(* IEC 61131-3 sources: brdkVision/export/brdkViBase/V1.00.3, 2 files *)

(* ---- Types.typ ---- *)
TYPE
	brdkViBase_hw_in_common_typ : 	STRUCT  (*B&R common hardware input structure from device*)
		hardwareVariant : UDINT; (*The hardware variant of the module can be read from this data point.*)
		moduleId : UDINT; (*The module hardware ID used to determine the type of device that can be read from this register. This is also listed in the respective technical data as the "B&R ID code". In addition, a serial number is printed on each module; the module hardware ID corresponds to the first four positions of this serial number.*)
		firmwareVersion : UDINT; (*The firmware version of the module can be read from this data point.
The last two positions correspond to the number after the decimal point.
Example: 345 corresponds to version 3.45.*)
		serialNumber : UDINT; (*The module's unique serial number can be read from this register. This 7-digit serial number is printed in decimal form on the module's housing*)
		moduleOk : BOOL; (*Status bit that indicates whether the module is physically present and configured. Detection takes place via the Fieldbus connection.*)
	END_STRUCT;
	brdkViBase_2d_typ : 	STRUCT  (*2D vector information.*)
		y : LREAL; (*Y-coordinate.*)
		x : LREAL; (*X-coordinate.*)
	END_STRUCT;
	brdkViBase_3d_typ : 	STRUCT  (*3D vector information.*)
		y : LREAL; (*Y-coordinate.*)
		z : LREAL; (*Z-coordinate.*)
		x : LREAL; (*X-coordinate.*)
	END_STRUCT;
	brdkViBase_angle_enum :
		( (*Angle enumeration type.*)
		BRDKVIBASE_ANGLE_X, (*X-angle*)
		BRDKVIBASE_ANGLE_Y, (*Y-angle*)
		BRDKVIBASE_ANGLE_Z (*Z-angle*)
		);
END_TYPE

(*Hw for camera *)

TYPE
	brdkViBase_cam_hw_out_typ : 	STRUCT  (*Camera hardware output structure to device*)
		par : brdkViBase_cam_hw_out_par_typ; (*Hardware output parameters to the device*)
		cmd : brdkViBase_cam_hw_out_cmd_typ; (*Hardware out commands to the device*)
	END_STRUCT;
	brdkViBase_cam_hw_out_cmd_typ : 	STRUCT  (*Camera hardware command structure to device*)
		imageAcquisition : BOOL; (*Enables/Disables the trigger for the image acquisition*)
		resetAcquisiton : BOOL; (*Cancels an image acquisition triggered by NetTime*)
		searchAcquisitonSettings : BOOL; (*Enables/Disables search for focus and integration time of the sensor*)
		digitalOutput : BOOL; (*Selects the mode of operation of the digital output*)
	END_STRUCT;
	brdkViBase_cam_hw_out_par_typ : 	STRUCT  (*Camera hardware parameter structure to device*)
		statusLED : USINT; (*Selects the mode and color of the LED status indicator bars. Constants BRDKVIBASE_STATUS_xxx can be used to set the color*)
		gainLevel : USINT; (*Sets a gain factor*)
		focus : UINT; (*Sets the focus from "MOD" to "Infinity", Unit depends on the selected one in the vision application file (um, mm, raw)*)
		exposureTime : UDINT; (*Sets the integration time of the sensor in microseconds*)
		flashColor : USINT; (*Selects LED colors of the onboard LED lighting. The constants BRDKVIBASE_LED_xxx can be used to set the color*)
		flashSegment : USINT; (*Enables/Disables LED segments. Binary patter for enable each of the four segments 0000 = all off, 1111 = all on*)
		chromaticLock : BOOL; (*Enables/Disables ChromaticLock*)
		IRFilter : BOOL; (*Enables/Disables the infrared filter*)
		delayNetTime : DINT; (*Sets Delay or NetTime for the trigger in microseconds*)
		cyclicLineScanPeriod : DINT; (*Time between 2 image acquisitions in dynamic line sensor operation.*)
		cyclicLineScanNettime : DINT; (*Specifies the NetTime for dynamic line sensor mode.*)
	END_STRUCT;
	brdkViBase_cam_hw_in_status_typ : 	STRUCT  (*Camera hardware status input structure from device*)
		sensorTemperature : SINT; (*Current camera temperature in °C*)
		lightWarningCnt : USINT; (*Counter for errors or warnings that have occurred related to lighting.*)
		cameraStatus : UDINT; (*This parameter specifies the status of the camera.*)
		acceptedAcquisitionCnt : USINT; (*Counter for accepted image acquisitions*)
		completedAcquisitionCnt : USINT; (*Counter for performed image acquisitions*)
		failedAcquisitionCnt : USINT; (*Counter for failed image acquisitions*)
		undervoltageError : BOOL; (*Power supply alarm*)
		imageAcquisitionReady : BOOL; (*Camera availability status*)
		imageProcessingActive : BOOL; (*Status of image processing execution *)
		digitalOutputStatus : BOOL; (*Status of digital output 01*)
		cameraProcessingTime : UINT; (*Processing time in milliseconds*)
		imageProcessingError : UINT; (*Bit pattern for displaying errors and warnings that occurred during image processing.*)
		imageNettime : DINT; (*NetTime of the image in microseconds*)
		digitalInput : BOOL; (*Status digital input (trigger input)*)
		gainLevel : USINT; (*Current GainLevel*)
		focus : UINT; (*Current focus setting from "MOD" to "Infinity", Unit depends on the selected one in the vision application file (um, mm, raw)*)
		exposureTime : UDINT; (*Current integration time of the sensor in microseconds *)
	END_STRUCT;
	brdkViBase_cam_hw_in_typ : 	STRUCT  (*Camera hardware input structure from device*)
		common : brdkViBase_hw_in_common_typ; (*B&R Hardware common inputs from device*)
		status : brdkViBase_cam_hw_in_status_typ; (*Camera hardware status inputs from device*)
	END_STRUCT;
	brdkViBase_cam_hw_typ : 	STRUCT  (*Camera hardware structure*)
		in : brdkViBase_cam_hw_in_typ; (*Camera hardware inputs from device*)
		out : brdkViBase_cam_hw_out_typ; (*Camera hardware outputs to device*)
	END_STRUCT;
END_TYPE

(*hw for light*)

TYPE
	brdkViBase_light_hw_out_typ : 	STRUCT  (*Light hardware output structure to device*)
		cmd : brdkViBase_light_hw_out_cmd_typ; (*Light hardware output commands to device*)
		par : brdkViBase_light_hw_out_par_typ; (*Light hardware output parameters to device*)
	END_STRUCT;
	brdkViBase_light_hw_status_typ : 	STRUCT  (*Light hardware status structure from device*)
		ready : BOOL; (*Lighting unit availability status*)
		status : UDINT; (*This parameter specifies the status of the lighting unit.*)
		acceptedFlashCnt : USINT; (*Counter for accepted lighting jobs*)
		completedFlashCnt : USINT; (*Counter for executed lighting jobs*)
		failedFlashCnt : USINT; (*Counter for failed lighting jobs*)
		LightWarningCnt : USINT; (*Counter for errors or warnings that have occurred related to lighting.*)
		sensorTemperature : SINT; (*Current lighting unit temperature in °C*)
	END_STRUCT;
	brdkViBase_light_hw_in_typ : 	STRUCT  (*Light hardware input structure from device*)
		common : brdkViBase_hw_in_common_typ; (*B&R hardware common inputs from device*)
		status : brdkViBase_light_hw_status_typ; (*Light hardware status inputs from device*)
	END_STRUCT;
	brdkViBase_light_hw_typ : 	STRUCT  (*Light hardware structure*)
		in : brdkViBase_light_hw_in_typ; (*Light hardware inputs from device*)
		out : brdkViBase_light_hw_out_typ; (*Light hardware outputs to device*)
	END_STRUCT;
	brdkViBase_light_hw_out_cmd_typ : 	STRUCT  (*Light hardware output commands to device*)
		flashTrigger : BOOL; (*Enables/Disables the trigger for the lighting job*)
		resetFlashTrigger : BOOL; (*Canceling a lighting job triggered by NetTime*)
	END_STRUCT;
	brdkViBase_light_hw_out_par_typ : 	STRUCT  (*Light hardware parameter output structure to device*)
		flashColor : USINT; (*Select LED colors of the LED lighting
 Constant BRDKVIBASE_LED_xxx can be used to set the color*)
		exposureTime : UDINT; (*Sets the exposure time in µs*)
		flashAngle : USINT; (*Only for Lightbar. Position of the stepper motor in degree 0 to 135*)
		flashSegments : USINT; (*Only for Lightbar. Enables/Disables LED segments*)
		cyclicLineScanPeriod : DINT; (*Time between 2 flashes in dynamic line sensor operation.*)
		cyclicLineScanNettime : DINT; (*Specifies the NetTime for dynamic line sensor mode.*)
		nettime : DINT; (*Sets the NetTime for the trigger in µs*)
	END_STRUCT;
END_TYPE

(*hw for vision function*)

TYPE
	brdkviBase_hw_vf_out_offset_typ : 	STRUCT  (*Offset ROI outputs for vision functions*)
		x : DINT; (*Offset of the ROI in the x-direction in 1/100 pixel increments.*)
		y : DINT; (*Offset of the ROI in the y-direction in increments of 1/100 pixel.*)
		orientation : INT; (*Offset to orient the ROI from -179.99° to +180° in 1/100 degree steps*)
		rotCenterX : DINT; (*Offset to orient the ROI from -179.99° to +180° in 1/100 degree steps*)
		rotCenterY : DINT; (*Offset of the rotation center in the y-direction in increments of 1/100 pixel.*)
	END_STRUCT;
	brdkViBase_hw_vf_in_common_typ : 	STRUCT  (*Common vision function hardware input structure from device*)
		numResults : USINT; (*Number of results found*)
		functionProcessingTime : UINT; (*Processing time of the visual function in microseconds*)
	END_STRUCT;
	brdkViBase_hw_vf_out_common_typ : 	STRUCT  (*vision function hardware output structure to device*)
		enable : BOOL; (*Enables/Disables the function*)
		numSearchMax : USINT; (*Maximum number of codes to search*)
		alignment : USINT; (*0 = "None"
1 = "SetReference"
2 = "GenerateAlignmentData" *)
		offsetROI : brdkviBase_hw_vf_out_offset_typ; (*Offset ROI parameters*)
	END_STRUCT;
END_TYPE

(*VF BLOB*)

TYPE
	brdkViBase_hw_blob_out_typ : 	STRUCT  (*BLOB hardware output structure*)
		regionFeatures : BOOL; (*Enables the geometric exclusion procedure *)
		enhancedBlobInformation : BOOL; (*0 = Additional information is transferred (default).
1 = Additional information is not transferred.
Means an increase of FunctionProcessingTime *)
		common : brdkViBase_hw_vf_out_common_typ; (*Common vision function output*)
	END_STRUCT;
	brdkViBase_hw_blob_in_typ : 	STRUCT  (*BLOB hardware structure for a result*)
		modelNumber : USINT; (*ModelNumber of the found blob*)
		meanGreyValue : USINT; (*Arithmetic mean of grayscale values for the blob*)
		clipped : BOOL; (* Edge contact detection *)
		area : UDINT; (* Size (area) in pixels in increments of 1/100 pixel*)
		length : UDINT; (* Length of the found blob*)
		width : UDINT; (* Width of the found blob. Is always the longer of the two sides*)
		xMin : DINT; (* Extreme value in the column direction
Minimum column position of the BLOB area*)
		xMax : DINT; (*Extreme value in the column direction
Maximum column position of the BLOB area*)
		yMin : DINT; (*Extreme value in the line direction
Minimum line position of the BLOB area*)
		yMax : DINT; (*Extreme value in the line direction
Maximum line position of the BLOB area*)
		circularity : USINT; (*Circularity of the found blob in %*)
		rectangularity : USINT; (*Rectangularity of the found blob in %*)
		anisometry : UINT; (*Anisometry of the found blob*)
		innterCirclePositionX : DINT; (*Output of position X of the center point of the inner circle of the found blob determined by the algorithm in 1/100 pixels.*)
		innterCirclePositionY : DINT; (*Output of position Y of the center point of the inner circle of the found blob determined by the algorithm in 1/100 pixels.*)
		innterCircleRadius : UDINT; (*Output of the radius of the inner circle of the found blob determined by the algorithm in 1/100 pixels.*)
		positionX : DINT; (*X-position (of the found blob) in the image in increments of 1/100 pixel*)
		positionY : DINT; (*Y-position (of the found blob) in the image in increments of 1/100 pixel*)
		orientation : INT; (*-179.99° to +180° in increments of 1/100 degree*)
		rotCenterX : DINT; (*The value deviating from the specified taught-in Alignment model is output here. In 1/100 pixel steps*)
		rotCenterY : DINT; (*The value deviating from the specified taught-in Alignment model is output here. In 1/100 pixel steps*)
	END_STRUCT;
	brdkViBase_hw_blob_1_in_typ : 	STRUCT  (*BLOB hardware input structure for 1 BLOB result*)
		common : brdkViBase_hw_vf_in_common_typ;
		results : brdkViBase_hw_blob_in_typ;
	END_STRUCT;
	brdkViBase_hw_blob_1_typ : 	STRUCT  (*BLOB hardware structure for 1 BLOB result*)
		in : brdkViBase_hw_blob_1_in_typ;
		out : brdkViBase_hw_blob_out_typ;
	END_STRUCT;
	brdkViBase_hw_blob_10_in_typ : 	STRUCT  (*BLOB hardware input structure for 10 BLOB result*)
		common : brdkViBase_hw_vf_in_common_typ;
		results : ARRAY[0..9]OF brdkViBase_hw_blob_in_typ;
	END_STRUCT;
	brdkViBase_hw_blob_10_typ : 	STRUCT  (*BLOB hardware structure for 10 BLOB result*)
		in : brdkViBase_hw_blob_10_in_typ;
		out : brdkViBase_hw_blob_out_typ;
	END_STRUCT;
	brdkViBase_hw_blob_50_in_typ : 	STRUCT  (*BLOB hardware input structure for 50 BLOB result*)
		common : brdkViBase_hw_vf_in_common_typ;
		results : ARRAY[0..49]OF brdkViBase_hw_blob_in_typ;
	END_STRUCT;
	brdkViBase_hw_blob_50_typ : 	STRUCT  (*BLOB hardware structure for 50 BLOB result*)
		in : brdkViBase_hw_blob_10_in_typ;
		out : brdkViBase_hw_blob_out_typ;
	END_STRUCT;
	brdkViBase_hw_blob_100_in_typ : 	STRUCT  (*BLOB hardware input structure for 100 BLOB result*)
		common : brdkViBase_hw_vf_in_common_typ;
		results : ARRAY[0..99]OF brdkViBase_hw_blob_in_typ;
	END_STRUCT;
	brdkViBase_hw_blob_100_typ : 	STRUCT  (*BLOB hardware structure for 100 BLOB result*)
		in : brdkViBase_hw_blob_100_in_typ;
		out : brdkViBase_hw_blob_out_typ;
	END_STRUCT;
	brdkViBase_hw_blob_150_in_typ : 	STRUCT  (*BLOB hardware input structure for 150 BLOB result*)
		common : brdkViBase_hw_vf_in_common_typ;
		results : ARRAY[0..149]OF brdkViBase_hw_blob_in_typ;
	END_STRUCT;
	brdkViBase_hw_blob_150_typ : 	STRUCT  (*BLOB hardware structure for 150 BLOB result*)
		in : brdkViBase_hw_blob_150_in_typ;
		out : brdkViBase_hw_blob_out_typ;
	END_STRUCT;
	brdkViBase_hw_blob_200_in_typ : 	STRUCT  (*BLOB hardware input structure for 200 BLOB result*)
		common : brdkViBase_hw_vf_in_common_typ;
		results : ARRAY[0..199]OF brdkViBase_hw_blob_in_typ;
	END_STRUCT;
	brdkViBase_hw_blob_200_typ : 	STRUCT  (*BLOB hardware structure for 200 BLOB result*)
		in : brdkViBase_hw_blob_200_in_typ;
		out : brdkViBase_hw_blob_out_typ;
	END_STRUCT;
	brdkViBase_hw_blob_250_in_typ : 	STRUCT  (*BLOB hardware input structure for 250 BLOB result*)
		common : brdkViBase_hw_vf_in_common_typ;
		results : ARRAY[0..249]OF brdkViBase_hw_blob_in_typ;
	END_STRUCT;
	brdkViBase_hw_blob_250_typ : 	STRUCT  (*BLOB hardware structure for 250 BLOB result*)
		in : brdkViBase_hw_blob_250_in_typ;
		out : brdkViBase_hw_blob_out_typ;
	END_STRUCT;
END_TYPE

(*VF match*)

TYPE
	brdkViBase_hw_match_out_typ : 	STRUCT  (*Matching hardware output structure*)
		timeout : UINT; (*Time limit for the search time in increments of 1 ms. 0 = no timeout*)
		minScore : USINT; (*Minimum grade in percent as to whether a found object is accepted as a match.*)
		maxOverlap : USINT; (*Maximum degree of overlap in percent that found objects are permitted to have.*)
		common : brdkViBase_hw_vf_out_common_typ; (*Common vision function output*)
	END_STRUCT;
	brdkViBase_hw_match_in_typ : 	STRUCT  (*Matching hardware structure for a result*)
		modelNumber : USINT; (*ID/Number of the learned model (which matches the hit)*)
		score : USINT; (*Grade (quality score) of the Matching result concerning the model in the range of values from 0.0 to 1.0. In 1/100*)
		scale : USINT; (*For shape-based Matching. Scaling factor from 0.01 to 2.55 in increments of 0.01.*)
		positionX : DINT; (*X-position (of the found object) in the image in increments of 1/100 pixel*)
		positionY : DINT; (*Y-position (of the found object) in the image in increments of 1/100 pixel*)
		orientation : INT; (*-179.99° to +180° in increments of 1/100 degree*)
		rotCenterX : DINT; (*The value deviating from the specified taught-in Alignment model is output here. In 1/100 pixel steps.*)
		rotCenterY : DINT; (*The value deviating from the specified taught-in Alignment model is output here. In 1/100 pixel steps.*)
	END_STRUCT;
	brdkViBase_hw_match_1_in_typ : 	STRUCT  (*Matching hardware input structure for 1 result*)
		common : brdkViBase_hw_vf_in_common_typ;
		results : brdkViBase_hw_match_in_typ;
	END_STRUCT;
	brdkViBase_hw_match_1_typ : 	STRUCT  (*Matching hardware structure for 1 result*)
		in : brdkViBase_hw_match_1_in_typ;
		out : brdkViBase_hw_match_out_typ;
	END_STRUCT;
	brdkViBase_hw_match_10_in_typ : 	STRUCT  (*Matching hardware input structure for 10 results*)
		common : brdkViBase_hw_vf_in_common_typ;
		results : ARRAY[0..9]OF brdkViBase_hw_match_in_typ;
	END_STRUCT;
	brdkViBase_hw_match_10_typ : 	STRUCT  (*Matching hardware structure for 10 results*)
		in : brdkViBase_hw_match_10_in_typ;
		out : brdkViBase_hw_match_out_typ;
	END_STRUCT;
	brdkViBase_hw_match_50_in_typ : 	STRUCT  (*Matching hardware input structure for 50 results*)
		common : brdkViBase_hw_vf_in_common_typ;
		results : ARRAY[0..49]OF brdkViBase_hw_match_in_typ;
	END_STRUCT;
	brdkViBase_hw_match_50_typ : 	STRUCT  (*Matching hardware structure for 50 results*)
		in : brdkViBase_hw_match_50_in_typ;
		out : brdkViBase_hw_match_out_typ;
	END_STRUCT;
	brdkViBase_hw_match_100_in_typ : 	STRUCT  (*Matching hardware input structure for 100 results*)
		common : brdkViBase_hw_vf_in_common_typ;
		results : ARRAY[0..99]OF brdkViBase_hw_match_in_typ;
	END_STRUCT;
	brdkViBase_hw_match_100_typ : 	STRUCT  (*Matching hardware structure for 100 results*)
		in : brdkViBase_hw_match_100_in_typ;
		out : brdkViBase_hw_match_out_typ;
	END_STRUCT;
	brdkViBase_hw_match_150_in_typ : 	STRUCT  (*Matching hardware input structure for 150 results*)
		common : brdkViBase_hw_vf_in_common_typ;
		results : ARRAY[0..149]OF brdkViBase_hw_match_in_typ;
	END_STRUCT;
	brdkViBase_hw_match_150_typ : 	STRUCT  (*Matching hardware structure for 150 results*)
		in : brdkViBase_hw_match_150_in_typ;
		out : brdkViBase_hw_match_out_typ;
	END_STRUCT;
	brdkViBase_hw_match_200_in_typ : 	STRUCT  (*Matching hardware input structure for 200 results*)
		common : brdkViBase_hw_vf_in_common_typ;
		results : ARRAY[0..199]OF brdkViBase_hw_match_in_typ;
	END_STRUCT;
	brdkViBase_hw_match_200_typ : 	STRUCT  (*Matching hardware structure for 200 results*)
		in : brdkViBase_hw_match_200_in_typ;
		out : brdkViBase_hw_match_out_typ;
	END_STRUCT;
	brdkViBase_hw_match_250_in_typ : 	STRUCT  (*Matching hardware input structure for 250 results*)
		common : brdkViBase_hw_vf_in_common_typ;
		results : ARRAY[0..249]OF brdkViBase_hw_match_in_typ;
	END_STRUCT;
	brdkViBase_hw_match_250_typ : 	STRUCT  (*Matching hardware structure for 250 results*)
		in : brdkViBase_hw_match_250_in_typ;
		out : brdkViBase_hw_match_out_typ;
	END_STRUCT;
END_TYPE

(*VF OCR [50]*)

TYPE
	brdkViBase_hw_OCR_out_typ : 	STRUCT  (*OCR hardware output structure*)
		timeout : UINT; (*Time limit for the search time in increments of 1 ms. 0 = no timeout*)
		parameterMode : USINT; (*Selects predefined parameter sets*)
		grading : BOOL; (*Enables/Disables quality grading of the characters read.*)
		common : brdkViBase_hw_vf_out_common_typ; (*Common vision function output*)
	END_STRUCT;
	brdkViBase_hw_OCR_in_typ : 	STRUCT  (*OCR hardware input structure for a result with length 50*)
		data : STRING[50]; (*A tuple of classification results, e.g. ["2", "6", "1", "2"], size 50*)
		gradingValue : USINT; (*Probability for all segmented characters (minimum confidence of all characters in a line)*)
		positionX : DINT; (*X-position (of the found string) in the image in increments of 1/100 pixel*)
		positionY : DINT; (*Y-position (of the found string) in the image in increments of 1/100 pixel*)
		orientation : INT; (*-179.99° to +180° in increments of 1/100 degree*)
	END_STRUCT;
	brdkViBase_hw_OCR_1_in_typ : 	STRUCT  (*OCR hardware input structure for 1 result*)
		common : brdkViBase_hw_vf_in_common_typ;
		results : brdkViBase_hw_OCR_in_typ;
	END_STRUCT;
	brdkViBase_hw_OCR_1_typ : 	STRUCT  (*OCR hardware structure for 1 result*)
		in : brdkViBase_hw_OCR_1_in_typ;
		out : brdkViBase_hw_OCR_out_typ;
	END_STRUCT;
	brdkViBase_hw_OCR_10_in_typ : 	STRUCT  (*OCR hardware input structure for 10 results*)
		common : brdkViBase_hw_vf_in_common_typ;
		results : ARRAY[0..9]OF brdkViBase_hw_OCR_in_typ;
	END_STRUCT;
	brdkViBase_hw_OCR_10_typ : 	STRUCT  (*OCR hardware structure for 10 results*)
		in : brdkViBase_hw_OCR_10_in_typ;
		out : brdkViBase_hw_OCR_out_typ;
	END_STRUCT;
	brdkViBase_hw_OCR_50_in_typ : 	STRUCT  (*OCR hardware input structure for 50 results*)
		common : brdkViBase_hw_vf_in_common_typ;
		results : ARRAY[0..49]OF brdkViBase_hw_OCR_in_typ;
	END_STRUCT;
	brdkViBase_hw_OCR_50_typ : 	STRUCT  (*OCR hardware structure for 50 results*)
		in : brdkViBase_hw_OCR_50_in_typ;
		out : brdkViBase_hw_OCR_out_typ;
	END_STRUCT;
	brdkViBase_hw_OCR_100_in_typ : 	STRUCT  (*OCR hardware input structure for 100 results*)
		common : brdkViBase_hw_vf_in_common_typ;
		results : ARRAY[0..99]OF brdkViBase_hw_OCR_in_typ;
	END_STRUCT;
	brdkViBase_hw_OCR_100_typ : 	STRUCT  (*OCR hardware structure for 100 results*)
		in : brdkViBase_hw_OCR_100_in_typ;
		out : brdkViBase_hw_OCR_out_typ;
	END_STRUCT;
	brdkViBase_hw_OCR_150_in_typ : 	STRUCT  (*OCR hardware input structure for 150 results*)
		common : brdkViBase_hw_vf_in_common_typ;
		results : ARRAY[0..149]OF brdkViBase_hw_OCR_in_typ;
	END_STRUCT;
	brdkViBase_hw_OCR_150_typ : 	STRUCT  (*OCR hardware structure for 150 results*)
		in : brdkViBase_hw_OCR_150_in_typ;
		out : brdkViBase_hw_OCR_out_typ;
	END_STRUCT;
	brdkViBase_hw_OCR_200_in_typ : 	STRUCT  (*OCR hardware input structure for 200 results*)
		common : brdkViBase_hw_vf_in_common_typ;
		results : ARRAY[0..199]OF brdkViBase_hw_OCR_in_typ;
	END_STRUCT;
	brdkViBase_hw_OCR_200_typ : 	STRUCT  (*OCR hardware structure for 200 results*)
		in : brdkViBase_hw_OCR_200_in_typ;
		out : brdkViBase_hw_OCR_out_typ;
	END_STRUCT;
	brdkViBase_hw_OCR_250_in_typ : 	STRUCT  (*OCR hardware input structure for 250 results*)
		common : brdkViBase_hw_vf_in_common_typ;
		results : ARRAY[0..249]OF brdkViBase_hw_OCR_in_typ;
	END_STRUCT;
	brdkViBase_hw_OCR_250_typ : 	STRUCT  (*OCR hardware structure for 250 results*)
		in : brdkViBase_hw_OCR_250_in_typ;
		out : brdkViBase_hw_OCR_out_typ;
	END_STRUCT;
END_TYPE

(*VF PX*)

TYPE
	brdkViBase_hw_pxCnt_out_typ : 	STRUCT  (*PX counter hardware output structure*)
		enhancedPXInformation : BOOL; (*Enables/Disables transfer of additional information.
Has an influence on the processing time of the vision function.*)
		common : brdkViBase_hw_vf_out_common_typ; (*Common vision function output*)
	END_STRUCT;
	brdkViBase_hw_pxCnt_in_typ : 	STRUCT  (*PX counter hardware input structure for a result*)
		modelNumber : USINT; (*Model number of the result found*)
		numPixels : UDINT; (*Number of pixels that correspond to the configuration in the model*)
		minGray : USINT; (*Lowest grayscale value in the result*)
		maxGray : USINT; (*Highest grayscale value in the result*)
		meanGray : UINT; (*Arithmetic mean value of the grayscale values of the result*)
		deviationGray : UINT; (*Standard deviation of the grayscale values of the result*)
		medianGray : USINT; (*Median of the grayscale values of the result*)
		modelArea : UDINT; (*Size (area) of the model in pixels*)
		numConnectedComponents : UINT; (*Number of non-contiguous areas of the result*)
		positionX : DINT; (*X-position (center point) in the image in increments of 1/100 pixel*)
		positionY : DINT; (*Y-position (center point) in the image in increments of 1/100 pixel*)
	END_STRUCT;
	brdkViBase_hw_pxCnt_1_in_typ : 	STRUCT  (*PX counter hardware input structure for 1 result*)
		common : brdkViBase_hw_vf_in_common_typ;
		results : brdkViBase_hw_pxCnt_in_typ;
	END_STRUCT;
	brdkViBase_hw_pxCnt_1_typ : 	STRUCT  (*PX counter hardware structure for 1 result*)
		in : brdkViBase_hw_pxCnt_1_in_typ;
		out : brdkViBase_hw_pxCnt_out_typ;
	END_STRUCT;
	brdkViBase_hw_pxCnt_10_in_typ : 	STRUCT  (*PX counter hardware input structure for 10 results*)
		common : brdkViBase_hw_vf_in_common_typ;
		results : ARRAY[0..9]OF brdkViBase_hw_pxCnt_in_typ;
	END_STRUCT;
	brdkViBase_hw_pxCnt_10_typ : 	STRUCT  (*PX counter hardware structure for 10 results*)
		in : brdkViBase_hw_pxCnt_10_in_typ;
		out : brdkViBase_hw_pxCnt_out_typ;
	END_STRUCT;
	brdkViBase_hw_pxCnt_50_in_typ : 	STRUCT  (*PX counter hardware input structure for 50 results*)
		common : brdkViBase_hw_vf_in_common_typ;
		results : ARRAY[0..49]OF brdkViBase_hw_pxCnt_in_typ;
	END_STRUCT;
	brdkViBase_hw_pxCnt_50_typ : 	STRUCT  (*PX counter hardware structure for 50 results*)
		in : brdkViBase_hw_pxCnt_50_in_typ;
		out : brdkViBase_hw_pxCnt_out_typ;
	END_STRUCT;
	brdkViBase_hw_pxCnt_100_in_typ : 	STRUCT  (*PX counter hardware input structure for 100 results*)
		common : brdkViBase_hw_vf_in_common_typ;
		results : ARRAY[0..99]OF brdkViBase_hw_pxCnt_in_typ;
	END_STRUCT;
	brdkViBase_hw_pxCnt_100_typ : 	STRUCT  (*PX counter hardware structure for 100 results*)
		in : brdkViBase_hw_pxCnt_100_in_typ;
		out : brdkViBase_hw_pxCnt_out_typ;
	END_STRUCT;
	brdkViBase_hw_pxCnt_150_in_typ : 	STRUCT  (*PX counter hardware input structure for 150 results*)
		common : brdkViBase_hw_vf_in_common_typ;
		results : ARRAY[0..149]OF brdkViBase_hw_pxCnt_in_typ;
	END_STRUCT;
	brdkViBase_hw_pxCnt_150_typ : 	STRUCT  (*PX counter hardware structure for 150 results*)
		in : brdkViBase_hw_pxCnt_150_in_typ;
		out : brdkViBase_hw_pxCnt_out_typ;
	END_STRUCT;
	brdkViBase_hw_pxCnt_200_in_typ : 	STRUCT  (*PX counter hardware input structure for 200 results*)
		common : brdkViBase_hw_vf_in_common_typ;
		results : ARRAY[0..199]OF brdkViBase_hw_pxCnt_in_typ;
	END_STRUCT;
	brdkViBase_hw_pxCnt_200_typ : 	STRUCT  (*PX counter hardware structure for 200 results*)
		in : brdkViBase_hw_pxCnt_200_in_typ;
		out : brdkViBase_hw_pxCnt_out_typ;
	END_STRUCT;
	brdkViBase_hw_pxCnt_250_in_typ : 	STRUCT  (*PX counter hardware input structure for 250 results*)
		common : brdkViBase_hw_vf_in_common_typ;
		results : ARRAY[0..249]OF brdkViBase_hw_pxCnt_in_typ;
	END_STRUCT;
	brdkViBase_hw_pxCnt_250_typ : 	STRUCT  (*PX counter hardware structure for 250 results*)
		in : brdkViBase_hw_pxCnt_250_in_typ;
		out : brdkViBase_hw_pxCnt_out_typ;
	END_STRUCT;
END_TYPE

(*VF mes*)

TYPE
	brdkViBase_hw_mes_out_typ : 	STRUCT  (*Measurement hardware output structure*)
		common : brdkViBase_hw_vf_out_common_typ; (*Common vision function output*)
	END_STRUCT;
	brdkViBase_hw_mes_in_typ : 	STRUCT  (*Measurement hardware input structure for a result*)
		result : DINT; (*Measurement values. Depending on the operator, it is possible to return angle, orientation, length or distance values, or a combination of any of these in an array.*)
	END_STRUCT;
	brdkViBase_hw_mes_1_in_typ : 	STRUCT  (*Measurement hardware input structure for 1 result*)
		common : brdkViBase_hw_vf_in_common_typ;
		results : brdkViBase_hw_mes_in_typ;
	END_STRUCT;
	brdkViBase_hw_mes_1_typ : 	STRUCT  (*Measurement hardware structure for 1 result*)
		in : brdkViBase_hw_mes_1_in_typ;
		out : brdkViBase_hw_mes_out_typ;
	END_STRUCT;
	brdkViBase_hw_mes_10_in_typ : 	STRUCT  (*Measurement hardware input structure for 10 results*)
		common : brdkViBase_hw_vf_in_common_typ;
		results : ARRAY[0..9]OF brdkViBase_hw_mes_in_typ;
	END_STRUCT;
	brdkViBase_hw_mes_10_typ : 	STRUCT  (*Measurement hardware structure for 10 results*)
		in : brdkViBase_hw_mes_10_in_typ;
		out : brdkViBase_hw_mes_out_typ;
	END_STRUCT;
	brdkViBase_hw_mes_50_in_typ : 	STRUCT  (*Measurement hardware input structure for 50 results*)
		common : brdkViBase_hw_vf_in_common_typ;
		results : ARRAY[0..49]OF brdkViBase_hw_mes_in_typ;
	END_STRUCT;
	brdkViBase_hw_mes_50_typ : 	STRUCT  (*Measurement hardware structure for 50 results*)
		in : brdkViBase_hw_mes_50_in_typ;
		out : brdkViBase_hw_mes_out_typ;
	END_STRUCT;
	brdkViBase_hw_mes_100_in_typ : 	STRUCT  (*Measurement hardware input structure for 100 results*)
		common : brdkViBase_hw_vf_in_common_typ;
		results : ARRAY[0..99]OF brdkViBase_hw_mes_in_typ;
	END_STRUCT;
	brdkViBase_hw_mes_100_typ : 	STRUCT  (*Measurement hardware structure for 100 results*)
		in : brdkViBase_hw_mes_100_in_typ;
		out : brdkViBase_hw_mes_out_typ;
	END_STRUCT;
	brdkViBase_hw_mes_150_in_typ : 	STRUCT  (*Measurement hardware input structure for 150 results*)
		common : brdkViBase_hw_vf_in_common_typ;
		results : ARRAY[0..149]OF brdkViBase_hw_mes_in_typ;
	END_STRUCT;
	brdkViBase_hw_mes_150_typ : 	STRUCT  (*Measurement hardware structure for 150 results*)
		in : brdkViBase_hw_mes_150_in_typ;
		out : brdkViBase_hw_mes_out_typ;
	END_STRUCT;
	brdkViBase_hw_mes_200_in_typ : 	STRUCT  (*Measurement hardware input structure for 200 results*)
		common : brdkViBase_hw_vf_in_common_typ;
		results : ARRAY[0..199]OF brdkViBase_hw_mes_in_typ;
	END_STRUCT;
	brdkViBase_hw_mes_200_typ : 	STRUCT  (*Measurement hardware structure for 200 results*)
		in : brdkViBase_hw_mes_200_in_typ;
		out : brdkViBase_hw_mes_out_typ;
	END_STRUCT;
	brdkViBase_hw_mes_250_in_typ : 	STRUCT  (*Measurement hardware input structure for 250 results*)
		common : brdkViBase_hw_vf_in_common_typ;
		results : ARRAY[0..249]OF brdkViBase_hw_mes_in_typ;
	END_STRUCT;
	brdkViBase_hw_mes_250_typ : 	STRUCT  (*Measurement hardware structure for 250 results*)
		in : brdkViBase_hw_mes_250_in_typ;
		out : brdkViBase_hw_mes_out_typ;
	END_STRUCT;
END_TYPE

(*VF cr [50]*)

TYPE
	brdkViBase_hw_cr_out_typ : 	STRUCT  (*Code reader hardware output structure*)
		timeout : UINT; (*Time limit for the search time in increments of 1 ms. 0 = no timeout*)
		parameterOptimization : USINT; (*Automatically enables, disables or resets taught-in parameters*)
		parameterMode : USINT; (*Selects predefined parameter sets*)
		codeGrading : BOOL; (*Enables/Disables quality grading of the codes read.*)
		symbolType : USINT; (*Selects the code type to be searched for*)
		enableRobustness : BOOL; (*Enables/Disables robustness for the search of the selected code type*)
		common : brdkViBase_hw_vf_out_common_typ; (*Common vision function output*)
	END_STRUCT;
	brdkViBase_hw_cr_in_typ : 	STRUCT  (*Code Reader hardware input structure for a result*)
		data : STRING[50]; (*Returns the content of the found code as array OCTET.  Size 50*)
		symbolType : USINT; (*Symbol type of codes found.*)
		gradingValue : BOOL; (*Evaluation of the codes in terms of quality*)
		enhancedGradingInformation : STRING[23]; (*Output of extended grading information from which the general GradingValue assessment parameter is composed.*)
		positionX : DINT; (*X-position (of the found code) in the image in increments of 1/100 pixel.*)
		positionY : DINT; (*Y-position (of the found code) in the image in increments of 1/100 pixel.*)
		orientation : INT; (*179.99° to +180° in increments of 1/100 degree*)
		rotCenterX : DINT; (*The value deviating from the specified taught-in Alignment model is output here. In 1/100 pixel steps.*)
		rotCenterY : DINT; (*The value deviating from the specified taught-in Alignment model is output here. In 1/100 pixel steps.*)
	END_STRUCT;
	brdkViBase_hw_cr_1_in_typ : 	STRUCT  (*Code reader hardware structure for 1 result*)
		common : brdkViBase_hw_vf_in_common_typ;
		results : brdkViBase_hw_cr_in_typ;
	END_STRUCT;
	brdkViBase_hw_cr_1_typ : 	STRUCT  (*Code reader hardware structure for 1 result*)
		in : brdkViBase_hw_cr_1_in_typ;
		out : brdkViBase_hw_cr_out_typ;
	END_STRUCT;
	brdkViBase_hw_cr_10_in_typ : 	STRUCT  (*Code reader hardware input structure for 10 results*)
		common : brdkViBase_hw_vf_in_common_typ;
		results : ARRAY[0..9]OF brdkViBase_hw_cr_in_typ;
	END_STRUCT;
	brdkViBase_hw_cr_10_typ : 	STRUCT  (*Code reader hardware structure for 10 results*)
		in : brdkViBase_hw_cr_10_in_typ;
		out : brdkViBase_hw_cr_out_typ;
	END_STRUCT;
	brdkViBase_hw_cr_50_in_typ : 	STRUCT  (*Code reader hardware input structure for 50 results*)
		common : brdkViBase_hw_vf_in_common_typ;
		results : ARRAY[0..49]OF brdkViBase_hw_cr_in_typ;
	END_STRUCT;
	brdkViBase_hw_cr_50_typ : 	STRUCT  (*Code reader hardware structure for 50 results*)
		in : brdkViBase_hw_cr_50_in_typ;
		out : brdkViBase_hw_cr_out_typ;
	END_STRUCT;
	brdkViBase_hw_cr_100_in_typ : 	STRUCT  (*Code reader hardware input structure for 100 results*)
		common : brdkViBase_hw_vf_in_common_typ;
		results : ARRAY[0..99]OF brdkViBase_hw_cr_in_typ;
	END_STRUCT;
	brdkViBase_hw_cr_100_typ : 	STRUCT  (*Code reader hardware structure for 100 results*)
		in : brdkViBase_hw_cr_100_in_typ;
		out : brdkViBase_hw_cr_out_typ;
	END_STRUCT;
	brdkViBase_hw_cr_150_in_typ : 	STRUCT  (*Code reader hardware input structure for 150 results*)
		common : brdkViBase_hw_vf_in_common_typ;
		results : ARRAY[0..149]OF brdkViBase_hw_cr_in_typ;
	END_STRUCT;
	brdkViBase_hw_cr_150_typ : 	STRUCT  (*Code reader hardware structure for 150 results*)
		in : brdkViBase_hw_cr_150_in_typ;
		out : brdkViBase_hw_cr_out_typ;
	END_STRUCT;
	brdkViBase_hw_cr_200_in_typ : 	STRUCT  (*Code reader hardware input structure for 200 results*)
		common : brdkViBase_hw_vf_in_common_typ;
		results : ARRAY[0..199]OF brdkViBase_hw_cr_in_typ;
	END_STRUCT;
	brdkViBase_hw_cr_200_typ : 	STRUCT  (*Code reader hardware structure for 200 results*)
		in : brdkViBase_hw_cr_200_in_typ;
		out : brdkViBase_hw_cr_out_typ;
	END_STRUCT;
	brdkViBase_hw_cr_250_in_typ : 	STRUCT  (*Code reader hardware input structure for 250 results*)
		common : brdkViBase_hw_vf_in_common_typ;
		results : ARRAY[0..249]OF brdkViBase_hw_cr_in_typ;
	END_STRUCT;
	brdkViBase_hw_cr_250_typ : 	STRUCT  (*Code reader hardware structure for 250 results*)
		in : brdkViBase_hw_cr_250_in_typ;
		out : brdkViBase_hw_cr_out_typ;
	END_STRUCT;
END_TYPE

(*VF sub*)

TYPE
	brdkViBase_hw_subBlob_out_typ : 	STRUCT  (*Subpixel BLOB hardware output structure *)
		regionFeatures : BOOL; (*Enables the geometric exclusion procedure *)
		enhancedBlobInformation : BOOL; (*0 = Additional information is transferred (default).
1 = Additional information is not transferred.
Means an increase of FunctionProcessingTime *)
		common : brdkViBase_hw_vf_out_common_typ; (*Common vision function output*)
	END_STRUCT;
	brdkViBase_hw_subBlob_in_typ : 	STRUCT  (*Subpixel BLOB hardware structure for a result*)
		modelNumber : USINT; (*ModelNumber of the found blob*)
		meanGreyValue : USINT; (*Arithmetic mean of grayscale values for the blob*)
		clipped : BOOL; (* Edge contact detection *)
		area : UDINT; (* Size (area) in pixels in increments of 1/100 pixel*)
		length : UDINT; (* Length of the found blob*)
		width : UDINT; (* Width of the found blob. Is always the longer of the two sides*)
		xMin : DINT; (* Extreme value in the column direction
Minimum column position of the BLOB area*)
		xMax : DINT; (*Extreme value in the column direction
Maximum column position of the BLOB area*)
		yMin : DINT; (*Extreme value in the line direction
Minimum line position of the BLOB area*)
		yMax : DINT; (*Extreme value in the line direction
Maximum line position of the BLOB area*)
		circularity : USINT; (*Circularity of the found blob in %*)
		rectangularity : USINT; (*Rectangularity of the found blob in %*)
		anisometry : UINT; (*Anisometry of the found blob*)
		innterCirclePositionX : DINT; (*Output of position X of the center point of the inner circle of the found blob determined by the algorithm in 1/100 pixels.*)
		innterCirclePositionY : DINT; (*Output of position Y of the center point of the inner circle of the found blob determined by the algorithm in 1/100 pixels.*)
		innterCircleRadius : UDINT; (*Output of the radius of the inner circle of the found blob determined by the algorithm in 1/100 pixels.*)
		positionX : DINT; (*X-position (of the found blob) in the image in increments of 1/100 pixel*)
		positionY : DINT; (*Y-position (of the found blob) in the image in increments of 1/100 pixel*)
		orientation : INT; (*-179.99° to +180° in increments of 1/100 degree*)
		rotCenterX : DINT; (*The value deviating from the specified taught-in Alignment model is output here. In 1/100 pixel steps*)
		rotCenterY : DINT; (*The value deviating from the specified taught-in Alignment model is output here. In 1/100 pixel steps*)
	END_STRUCT;
	brdkViBase_hw_subBlob_1_in_typ : 	STRUCT  (*Subpixel BLOB hardware input structure for 1 result*)
		common : brdkViBase_hw_vf_in_common_typ;
		results : brdkViBase_hw_subBlob_in_typ;
	END_STRUCT;
	brdkViBase_hw_subBlob_1_typ : 	STRUCT  (*Subpixel BLOB hardware structure for 1 result*)
		in : brdkViBase_hw_subBlob_1_in_typ;
		out : brdkViBase_hw_subBlob_out_typ;
	END_STRUCT;
	brdkViBase_hw_subBlob_10_in_typ : 	STRUCT  (*Subpixel BLOB hardware input structure for 10 results*)
		common : brdkViBase_hw_vf_in_common_typ;
		results : ARRAY[0..9]OF brdkViBase_hw_subBlob_in_typ;
	END_STRUCT;
	brdkViBase_hw_subBlob_10_typ : 	STRUCT  (*Subpixel BLOB hardware structure for 10 results*)
		in : brdkViBase_hw_subBlob_10_in_typ;
		out : brdkViBase_hw_subBlob_out_typ;
	END_STRUCT;
	brdkViBase_hw_subBlob_50_in_typ : 	STRUCT  (*Subpixel BLOB hardware input structure for 50 results*)
		common : brdkViBase_hw_vf_in_common_typ;
		results : ARRAY[0..49]OF brdkViBase_hw_subBlob_in_typ;
	END_STRUCT;
	brdkViBase_hw_subBlob_50_typ : 	STRUCT  (*Subpixel BLOB hardware structure for 50 results*)
		in : brdkViBase_hw_subBlob_50_in_typ;
		out : brdkViBase_hw_subBlob_out_typ;
	END_STRUCT;
	brdkViBase_hw_subBlob_100_in_typ : 	STRUCT  (*Subpixel BLOB hardware input structure for 100 results*)
		common : brdkViBase_hw_vf_in_common_typ;
		results : ARRAY[0..99]OF brdkViBase_hw_subBlob_in_typ;
	END_STRUCT;
	brdkViBase_hw_subBlob_100_typ : 	STRUCT  (*Subpixel BLOB hardware structure for 100 results*)
		in : brdkViBase_hw_subBlob_100_in_typ;
		out : brdkViBase_hw_subBlob_out_typ;
	END_STRUCT;
	brdkViBase_hw_subBlob_150_in_typ : 	STRUCT  (*Subpixel BLOB hardware input structure for 150 results*)
		common : brdkViBase_hw_vf_in_common_typ;
		results : ARRAY[0..149]OF brdkViBase_hw_subBlob_in_typ;
	END_STRUCT;
	brdkViBase_hw_subBlob_150_typ : 	STRUCT  (*Subpixel BLOB hardware structure for 150 results*)
		in : brdkViBase_hw_subBlob_150_in_typ;
		out : brdkViBase_hw_subBlob_out_typ;
	END_STRUCT;
	brdkViBase_hw_subBlob_200_in_typ : 	STRUCT  (*Subpixel BLOB hardware input structure for 200 results*)
		common : brdkViBase_hw_vf_in_common_typ;
		results : ARRAY[0..199]OF brdkViBase_hw_subBlob_in_typ;
	END_STRUCT;
	brdkViBase_hw_subBlob_200_typ : 	STRUCT  (*Subpixel BLOB hardware structure for 200 results*)
		in : brdkViBase_hw_subBlob_200_in_typ;
		out : brdkViBase_hw_subBlob_out_typ;
	END_STRUCT;
	brdkViBase_hw_subBlob_250_in_typ : 	STRUCT  (*Subpixel BLOB hardware input structure for 250 results*)
		common : brdkViBase_hw_vf_in_common_typ;
		results : ARRAY[0..249]OF brdkViBase_hw_subBlob_in_typ;
	END_STRUCT;
	brdkViBase_hw_subBlob_250_typ : 	STRUCT  (*Subpixel BLOB hardware structure for 250 results*)
		in : brdkViBase_hw_subBlob_250_in_typ;
		out : brdkViBase_hw_subBlob_out_typ;
	END_STRUCT;
	brdkViBase_imgTrigger_sim_typ : 	STRUCT
		enable : BOOL;
		imgProcessingDelay : TIME;
	END_STRUCT;
	brdkViBase_imgTrigger_local_typ : 	STRUCT
		state : USINT;
		oldNettime : DINT;
		oldAccCnt : USINT;
		initDone : BOOL;
		triggerActive : BOOL;
		simDelay : TON;
		waitForImage : BOOL;
	END_STRUCT;
END_TYPE

(* ---- brdkViBase.fun ---- *)
FUNCTION brdkViBase_distance : LREAL (*Calculate the distance between two points.*) (*$GROUP=User,$CAT=User,$GROUPICON=User.png,$CATICON=User.png*)
	VAR_INPUT
		x1 : LREAL; (*Point 1 x*)
		y1 : LREAL; (*Point 1 y*)
		x2 : LREAL; (*Point 2 x*)
		y2 : LREAL; (*Point 2 y*)
	END_VAR
END_FUNCTION

FUNCTION brdkViBase_random : INT (*Get a random number between min and max.*) (*$GROUP=User,$CAT=User,$GROUPICON=User.png,$CATICON=User.png*)
	VAR_INPUT
		min : INT; (*Min value*)
		max : INT; (*Max value*)
	END_VAR
END_FUNCTION

FUNCTION brdkViBase_initRand : BOOL (*Initialize rand function.*) (*$GROUP=User,$CAT=User,$GROUPICON=User.png,$CATICON=User.png*)
	VAR_INPUT
		seed : UDINT; (*seed*)
	END_VAR
END_FUNCTION

FUNCTION brdkViBase_deg2rad : LREAL (* Function to convert degrees to radians. Return angle in radians.*) (*$GROUP=User,$CAT=User,$GROUPICON=User.png,$CATICON=User.png*)
	VAR_INPUT
		deg : LREAL; (*Input degree.*)
	END_VAR
END_FUNCTION

FUNCTION brdkViBase_rad2deg : LREAL (*Function to convert radian to degree. Return angle in degrees.*) (*$GROUP=User,$CAT=User,$GROUPICON=User.png,$CATICON=User.png*)
	VAR_INPUT
		rad : LREAL; (*Input radian.*)
	END_VAR
END_FUNCTION

{REDUND_ERROR} FUNCTION_BLOCK brdkViBase_imgTrigger (*Function block to handle triggering of new image on a camera*) (*$GROUP=User,$CAT=User,$GROUPICON=User.png,$CATICON=User.png*)
	VAR_INPUT
		pCameraHw : REFERENCE TO brdkViBase_cam_hw_typ; (*Pointer to a brdkViBase Camera hardware stucture*)
		numLights : USINT; (*Number of lights used for this camera, if more than 1 then pLightHw need to be an array*)
		pLightHw : REFERENCE TO brdkViBase_light_hw_typ; (*Pointer to a brdkViBase light hardware structure, can also be an array of these structures*)
		searchAcquisitonSettings : BOOL; (*Start the search acquisition settings routine is done*)
		useCamColorForLight : BOOL; (*If true then the camera flash color is also used as flash color  on the lights*)
		useCamExpTimeForLight : BOOL; (*If true then the camera exposure time is also used as exposure time on the lights*)
		trigger : BOOL; (*Trigger a new image, is automatically reset*)
		delayNettime : DINT; (*Sets Delay or NetTime for the trigger in microseconds, is used in same cycle as trigger is true*)
		simulate : brdkViBase_imgTrigger_sim_typ; (*Simulation data structure, for configuring simulation of the function block*)
	END_VAR
	VAR_OUTPUT
		newImage : {REDUND_UNREPLICABLE} BOOL; (*New image results are ready, only high one cycle*)
		searchAcquisitonSettingsDone : BOOL; (*The search acquisition settings routine is done *)
		ready : {REDUND_UNREPLICABLE} BOOL; (*All devices are ready to receive a new trigger request*)
		hwError : BOOL; (*One or more devices are not present (moduleOk = false)*)
		busy : {REDUND_UNREPLICABLE} BOOL; (*Busy is true from image trigger to image result is returned*)
		imageResultCnt : UDINT; (*Number received image results*)
		triggerCnt : UDINT; (*Number of image acquisitions that have been accepted*)
	END_VAR
	VAR
		internal : brdkViBase_imgTrigger_local_typ;
	END_VAR
END_FUNCTION_BLOCK

{REDUND_ERROR} FUNCTION brdkViBase_LEDIntensity : UDINT (*Function to correct the LED intensity (exposure time) between different flash LED colors*) (*$GROUP=User,$CAT=User,$GROUPICON=User.png,$CATICON=User.png*)
	VAR_INPUT
		LEDLenseType : USINT; (*LED type 1, 2 or 3*)
		distance : UINT; (*Distance to the object in mm *)
		exposureTime : UDINT; (*exposure time of the fromColor*)
		fromColor : USINT; (*Flash LED color to convert from*)
		toColor : USINT; (*Flash LED color to convert to*)
	END_VAR
END_FUNCTION
